(* CODESYS project withopc.export

Project tree, tasks and I/O mapping:
  Device : CODESYS Control Win V3, 3S - Smart Software Solutions GmbH, version 3.5.18.40
    application Application
      libraries: Standard, 3.5.18.0 (System); VisuDialogs, * (System); SysTime, 3.5.17.0 (System)
      task MainTask (cyclic, interval 100 ms, priority 1) calls PLC_PRG, POU, POU_1
      task VISU_TASK (cyclic, interval 100 ms, priority 31) calls VisuElems.Visu_Prg
      Communication Manager
        OPC_UA_Symbols
          Information Model
      OPC_UA_Symbols Objects/
        function block fsmType [ST]
      program PLC_PRG [SFC]: Init_entry, Step0_entry, Step1_entry, Step2_active
      program POU [ST]
      program POU_1 [LD]
      visualisation Visualization
  text list GlobalTextList
*)

// Device/Application/PLC_PRG
PROGRAM PLC_PRG
VAR
	
{attribute 'opcua.mapping.member.accesslevel' := 'CurrentRead'}
	OnState : BOOL;
	{attribute 'opcua.mapping.member.accesslevel' := 'CurrentRead'}
	TotalTimeOn : LREAL;
	{attribute 'opcua.mapping.member.accesslevel' := 'CurrentRead'}
	RunningState : BOOL;

	{attribute 'opcua.mapping.member.accesslevel' := 'CurrentRead'}
	LastTimeRunning : ULINT;
	
	{attribute 'opcua.mapping.member.accesslevel' := 'CurrentRead'}
	Result : UDINT;
	udiUTC_DateAndTime : UDINT;
	udiLocal_DateAndTime : UDINT;
	LastTimeStop : ULINT;
	{attribute 'opcua.mapping.member.accesslevel' := 'CurrentRead'}
	machineType : STRING;
	pause: BOOL;
	start: BOOL;
	stop: BOOL;
	init_ok: BOOL;
	wt: TIME;
	Tinit: TON;
	warming: BOOL;

END_VAR

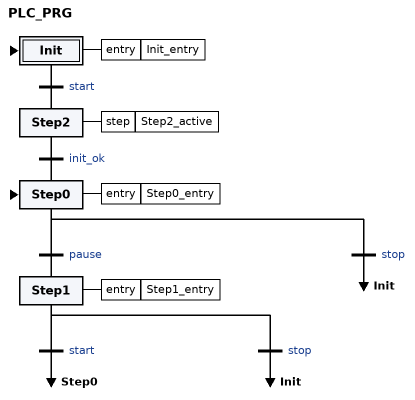
INITIAL_STEP Init:
    Init_entry(P1);  // entry action
END_STEP
TRANSITION FROM Init TO Step2
    := start;
END_TRANSITION
STEP Step2:
    Step2_active(N);  // step action
END_STEP
TRANSITION FROM Step2 TO Step0
    := init_ok;
END_TRANSITION
STEP Step0:
    Step0_entry(P1);  // entry action
END_STEP
TRANSITION FROM Step0 TO Step1
    := pause;
END_TRANSITION
STEP Step1:
    Step1_entry(P1);  // entry action
END_STEP
TRANSITION FROM Step0 TO Init
    := stop;
END_TRANSITION
TRANSITION FROM Step1 TO Step0
    := start;
END_TRANSITION
TRANSITION FROM Step1 TO Init
    := stop;
END_TRANSITION

ACTION Init_entry:
OnState := FALSE;
RunningState := FALSE;
END_ACTION

ACTION Step0_entry:
RunningState := TRUE;
warming := FALSE;
LastTimeRunning := TO_ULINT(SysTimeRtcGet(Result));
END_ACTION

ACTION Step1_entry:
RunningState := FALSE;
LastTimeStop := TO_ULINT(SysTimeRtcGet(Result));
END_ACTION

ACTION Step2_active:
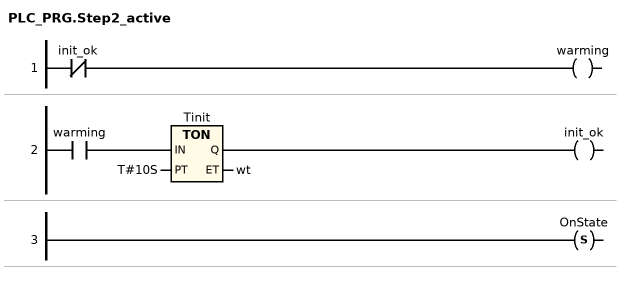
// NETWORK 1
warming := NOT init_ok;

// NETWORK 2
Tinit(IN := warming, PT := T#10S, ET => wt); // TON
init_ok := Tinit.Q;

// NETWORK 3
OnState S= TRUE;
END_ACTION

END_PROGRAM

// Device/Application/POU
PROGRAM POU
VAR
	TotalTimeOn : LREAL;
	maxTime : TIME := UDINT_TO_TIME(4294967295);
END_VAR

TotalTimeOn := TO_LREAL(POU_1.ton1.ET);
OPC_UA_Symbols.inst_2();

END_PROGRAM

// Device/Application/POU_1
PROGRAM POU_1
VAR
	elapsed: TIME;
	done: BOOL;
	ton1: TON;
END_VAR

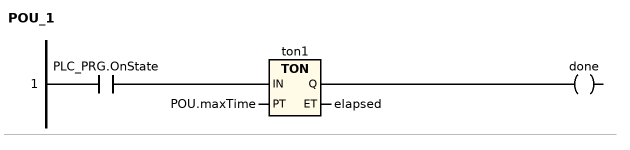
// NETWORK 1
ton1(IN := PLC_PRG.OnState, PT := POU.maxTime, ET => elapsed); // TON
done := ton1.Q;

END_PROGRAM

// Device/Application/OPC_UA_Symbols Objects/fsmType
{attribute 'opcua.mapping.type'}
{attribute 'opcua.mapping.modeluri' := 'http://opcfoundation.org/fsm'}
{attribute 'opcua.mapping.publicationdate' := '01/22/2023 00:00:00'}
{attribute 'opcua.mapping.nodeid' := 'nsu=http://opcfoundation.org/fsm;i=8'}
FUNCTION_BLOCK fsmType
VAR
	{attribute 'opcua.mapping.member.accesslevel' := 'CurrentRead'}
	OnState : BOOL;
	{attribute 'opcua.mapping.member.accesslevel' := 'CurrentRead'}
	TotalTimeOn : LREAL;
	{attribute 'opcua.mapping.member.accesslevel' := 'CurrentRead'}
	RunningState : BOOL;
// 	{attribute 'opcua.mapping.member.accesslevel' := 'CurrentRead'}
// 	TotalTimeRunning : LREAL;
	{attribute 'opcua.mapping.member.accesslevel' := 'CurrentRead'}
	LastTimeRunning : ULINT;
	{attribute 'opcua.mapping.member.accesslevel' := 'CurrentRead'}
	LastTimeStop : ULINT;
	{attribute 'opcua.mapping.member.accesslevel' := 'CurrentRead'}
	machineType : STRING;
END_VAR

OnState := PLC_PRG.OnState;
{attribute 'opcua.mapping.member.accesslevel' := 'CurrentRead'}
	{attribute 'opcua.mapping.member.accesslevel' := 'CurrentRead'}
RunningState := PLC_PRG.RunningState;
	{attribute 'opcua.mapping.member.accesslevel' := 'CurrentRead'}
// TotalTimeRunning;
// 	{attribute 'opcua.mapping.member.accesslevel' := 'CurrentRead'}
LastTimeRunning := PLC_PRG.LastTimeRunning;
	{attribute 'opcua.mapping.member.accesslevel' := 'CurrentRead'}
LastTimeStop := PLC_PRG.LastTimeStop;
	{attribute 'opcua.mapping.member.accesslevel' := 'CurrentRead'}
machineType := 'Simple FSM model';

TotalTimeOn :=  POU.TotalTimeOn;

END_FUNCTION_BLOCK

// Device/Application/Visualization
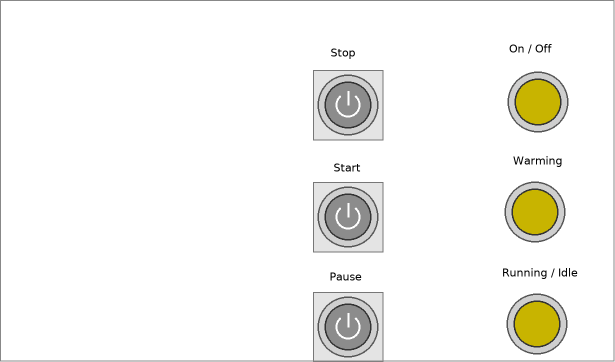
VISUALIZATION Visualization  // 615x362
    PowerSwitch (313,70 70x70), variable: PLC_PRG.stop, behaviour: TAP, style: Switch-PowerSwitch-Gray
    PowerSwitch (313,182 70x70), variable: PLC_PRG.start, behaviour: TAP, style: Switch-PowerSwitch-Gray
    PowerSwitch (313,292 70x70), variable: PLC_PRG.pause, behaviour: TAP, style: Switch-PowerSwitch-Gray
    Lamp1 (503,67 70x70), variable: PLC_PRG.OnState, style: Lamp-Lamp1-Yellow
    Lamp1 (502,289 70x70), variable: PLC_PRG.RunningState, style: Lamp-Lamp1-Yellow
    Label (268,38 150x30), "Stop"
    Label (272,153 150x30), "Start"
    Label (271,262 150x30), "Pause"
    Label (465,258 150x30), "Running / Idle"
    Label (454,33 153x32), "On / Off"
    Lamp1 (500,177 70x70), variable: PLC_PRG.warming, style: Lamp-Lamp1-Yellow
    Label (463,146 150x30), "Warming"
END_VISUALIZATION
